// TIA Portal project "Practica1" (V16)

(* hardware
DEVICE "S7-1200 station_1"  S7-1200 Station
   slot 0: "Rack_0"  S7-1200 Rack  Rack  V1.0
   slot 1: "PLC_1"  CPU 1214C AC/DC/Rly  6ES7 214-1BG40-0XB0  V4.2
*)

// ===== PLC "PLC_1"  CPU 1214C AC/DC/Rly =====

VAR_GLOBAL   // PLC tag table "Tabla de variables_1"
   "Marcha" AT %I0.0 : Bool;
   "Paro" AT %I0.1 : Bool;
   "Luz" AT %Q0.2 : Bool;
   "Interruptor" AT %I0.2 : Bool;
   "Luz(1)" AT %Q0.3 : Bool;
END_VAR

ORGANIZATION_BLOCK "Main"   // OB1, LAD, ProgramCycle
TITLE = "Main Program Sweep (Cycle)"
{ S7_Optimized_Access := 'TRUE' }
VERSION : 0.1
   VAR_INPUT
      Initial_Call : Bool;   // Initial call of this OB
      Remanence : Bool;   // =True, if remanent data are available
   END_VAR
BEGIN

REGION Network 1
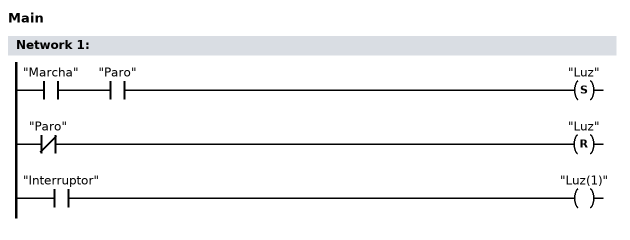
   RUNG wire#powerrail
      Contact( "Marcha" )
      Contact( "Paro" )
      S_Coil( "Luz" )
   END_RUNG
   RUNG wire#powerrail
      I_Contact( "Paro" )
      R_Coil( "Luz" )
   END_RUNG
   RUNG wire#powerrail
      Contact( "Interruptor" )
      Coil( "Luz(1)" )
   END_RUNG
   // the same network as SCL:
   IF "Marcha" AND "Paro" THEN "Luz" := TRUE; END_IF;
   IF NOT "Paro" THEN "Luz" := FALSE; END_IF;
   "Luz(1)" := "Interruptor";
END_REGION
END_ORGANIZATION_BLOCK